// TIA Portal V20 export
TYPE "typeCmHmiInterfaceSafeRef"
// stored: Access Published, Namespace Unit1.Em2
   STRUCT
      jrOutPnPLeftAxisY : "LER_typeSafeReferencingInterface";
      jrOutPnPLeftAxisZ : "LER_typeSafeReferencingInterface";
   END_STRUCT;
END_TYPE
